# EPICS substitutions: iocBoot/ioc6idACS1/substitutions/canberra_3.substitutions
file "$(MCA)/mcaApp/Db/simple_mca.db"
{
pattern
{P           M       DTYP           INP              PREC  CHANS}
{6idACS1:med:   mca1  "asynMCA"       "@asyn(AIM1/1 0)"  3     2048}
{6idACS1:med:   mca2  "asynMCA"       "@asyn(AIM1/2 0)"  3     2048}
{6idACS1:med:   mca3  "asynMCA"       "@asyn(AIM2/1 0)"  3     2048}
{6idACS1:med:   mca0  "Soft Channel"  ""                 3     2048}
}

#file "$(MCA)/mcaApp/Db/icb_amp.db"
#{
#pattern
#{P			AMP		PORT}
#{6idACS1:med:	amp1	icbAmp1}
#}

file "$(MCA)/mcaApp/Db/icb_adc.db"
{
pattern
{P			ADC		PORT}
{6idACS1:med:	adc1	"icbAdc1"}
{6idACS1:med:	adc2	"icbAdc2"}
{6idACS1:med:	adc3	"icbAdc3"}
}

#file "$(MCA)/mcaApp/Db/icb_hvps.db"
#{
#pattern
#{P			HVPS	LIMIT	PORT}
#{6idACS1:med:	hvps1	1000	"icbHvps1"}
#}

file "$(MCA)/mcaApp/Db/icb_tca.db"
{
pattern
{P,          TCA,	PORT,		MCA}
{6idACS1:med:,  tca1,	"icbTca1",	mca1}
{6idACS1:med:,  tca2,	"icbTca2",	mca2}
{6idACS1:med:,  tca3,	"icbTca3",	mca3}
}
